// TIA Portal V18 export
FUNCTION "DevTempGarb" : Void   // FC13, LAD
TITLE = Development garbarge area
{ S7_Optimized_Access := 'TRUE' }
AUTHOR : HenriP
VERSION : 0.1
// To use when removing part of the code for test
// stored: AutoNumber true, IsIECCheckEnabled false, SetENOAutomatically false, UDAEnableTagReadback false
BEGIN
END_FUNCTION
